TYPE ST_LeakTester_CMD :
STRUCT
	
	RunLeakTester1		: BOOL;		
	RunLeakTester2		: BOOL;	
	
END_STRUCT
END_TYPE

(* stored: Version 1.1.0.1, ProductVersion 3.1.4024.13
   DUT ST_LeakTester_CMD: Id {6505ec06-2249-4aa6-b866-f6c95a817053} *)
